// TwinCAT 3 PLC project XPlanarPLC
// ProgramVersion: 3.1.4026.19
// libraries:
//   SPT Base Types, * (Beckhoff Automation LLC)
//   Tc2_Standard, * (Beckhoff Automation GmbH)
//   Tc2_System, * (Beckhoff Automation GmbH)
//   Tc2_Utilities, * (Beckhoff Automation GmbH)
//   Tc3_Mc3PlanarMotion, * (Beckhoff Automation GmbH)
//   Tc3_XPlanarUtility, * (Beckhoff Automation GmbH)
//   XPlanarApplication, * (Beckhoff Automation LLC)
// project tree:
//   DUTs/Estop/ E_EStop.TcDUT, ST_EstopIO.TcDUT, U_Estop.TcDUT
//   DUTs/ E_DemoStep.TcDUT, ST_Point.TcDUT
//   DUTs/Selector switch/ E_SelectorSwitchPos.TcDUT, ST_SelectorSwitchIO.TcDUT, U_SelectorSwitch.TcDUT
//   / PlcTask.TcTTO
//   POUs/ F_SetAllMoversMovement.TcPOU, F_SetAllMoversRotation.TcPOU, MAIN.TcPOU
//   POUs/Pushbuttons/ FB_Pushbutton.TcPOU, LED_Color_Enum.TcDUT, Pushbutton_Enum.TcDUT
// real-time tasks:
//   TASK PlcTask: cycle T#10ms, priority 20, ADS port 350
//   TASK XPlanar Task3: cycle T#250us, priority 1, ADS port 351
//   TASK MC-Task (MET): cycle T#2ms, priority 2, ADS port 352
//   TASK MC-Task (MPT): cycle T#10ms, priority 3, ADS port 353
//   TASK Job Task: cycle default, priority 4
// I/O:
//   DEVICE Device 3 (EtherCAT), AmsNetId 172.18.232.79.4.1
//     Box 6 (PS2001-2420) [PS2001-2420-1001 Power supply (24V, 20A, 1-phase)]
//     Box 5 (EP2339-0003) [EP2339-0003 16 Ch. Dig. Input/Output 24V, 0,5A, 10-Pole Plug Connector]
//   DEVICE Device 1 (EtherCAT), AmsNetId 172.18.232.79.2.1
//     Term 1 (APS4322-7000) [APS4322-7000 Drive]
//       Term 2 (APS4322-5000) [APS4322-5000 Feedback]
//     Term 3 (APS4322-7000) [APS4322-7000 Drive]
//       Term 4 (APS4322-5000) [APS4322-5000 Feedback]
// variable links:
//   Device 1 (EtherCAT) <-> TcCOM Objects/XPlanar/Part1/Tile1
//     Term 3 (APS4322-7000)/APS Comm Inputs/CommStatusWord <-> Data Pointer/MoverCommStatusWord
//     Term 3 (APS4322-7000)/APS Comm Inputs/Data {1..4} <-> Data Pointer/MoverCommDataIn[{0..3}]  (4 links)
//     Term 3 (APS4322-7000)/APS Comm Outputs/CommControlWord <-> Data Pointer/MoverCommControlWord
//     Term 3 (APS4322-7000)/APS Comm Outputs/Data 1 <-> Data Pointer/MoverCommDataOut
//     Term 3 (APS4322-7000)/APS Diagdata/DC Link Voltage <-> Data Pointer/DcLinkVoltage
//     Term 3 (APS4322-7000)/APS Diagdata/Power supply current <-> Data Pointer/PowerSupplyCurrent
//     Term 3 (APS4322-7000)/APS Inputs/StatusWord <-> Data Pointer/PowerUnitStatusWord
//     Term 3 (APS4322-7000)/APS Outputs/ControlWord <-> Data Pointer/PowerUnitControlWord
//     Term 3 (APS4322-7000)/APS Outputs/Current D 0X0 <-> Data Pointer/DCurrentSetPoints[0]
//     Term 3 (APS4322-7000)/APS Outputs/Current D 0X1 <-> Data Pointer/DCurrentSetPoints[1]
//     Term 3 (APS4322-7000)/APS Outputs/Current D 0X2 <-> Data Pointer/DCurrentSetPoints[2]
//     Term 3 (APS4322-7000)/APS Outputs/Current D 1X0 <-> Data Pointer/DCurrentSetPoints[6]
//     Term 3 (APS4322-7000)/APS Outputs/Current D 1X1 <-> Data Pointer/DCurrentSetPoints[7]
//     Term 3 (APS4322-7000)/APS Outputs/Current D 1X2 <-> Data Pointer/DCurrentSetPoints[8]
//     Term 3 (APS4322-7000)/APS Outputs/Current D 2X0 <-> Data Pointer/DCurrentSetPoints[12]
//     Term 3 (APS4322-7000)/APS Outputs/Current D 2X1 <-> Data Pointer/DCurrentSetPoints[13]
//     Term 3 (APS4322-7000)/APS Outputs/Current D 2X2 <-> Data Pointer/DCurrentSetPoints[14]
//     Term 3 (APS4322-7000)/APS Outputs/Current D 3X0 <-> Data Pointer/DCurrentSetPoints[18]
//     Term 3 (APS4322-7000)/APS Outputs/Current D 3X1 <-> Data Pointer/DCurrentSetPoints[19]
//     Term 3 (APS4322-7000)/APS Outputs/Current D 3X2 <-> Data Pointer/DCurrentSetPoints[20]
//     Term 3 (APS4322-7000)/APS Outputs/Current D 0Y0 <-> Data Pointer/DCurrentSetPoints[3]
//     Term 3 (APS4322-7000)/APS Outputs/Current D 0Y1 <-> Data Pointer/DCurrentSetPoints[4]
//     Term 3 (APS4322-7000)/APS Outputs/Current D 0Y2 <-> Data Pointer/DCurrentSetPoints[5]
//     Term 3 (APS4322-7000)/APS Outputs/Current D 1Y0 <-> Data Pointer/DCurrentSetPoints[9]
//     Term 3 (APS4322-7000)/APS Outputs/Current D 1Y1 <-> Data Pointer/DCurrentSetPoints[10]
//     Term 3 (APS4322-7000)/APS Outputs/Current D 1Y2 <-> Data Pointer/DCurrentSetPoints[11]
//     Term 3 (APS4322-7000)/APS Outputs/Current D 2Y0 <-> Data Pointer/DCurrentSetPoints[15]
//     Term 3 (APS4322-7000)/APS Outputs/Current D 2Y1 <-> Data Pointer/DCurrentSetPoints[16]
//     Term 3 (APS4322-7000)/APS Outputs/Current D 2Y2 <-> Data Pointer/DCurrentSetPoints[17]
//     Term 3 (APS4322-7000)/APS Outputs/Current D 3Y0 <-> Data Pointer/DCurrentSetPoints[21]
//     Term 3 (APS4322-7000)/APS Outputs/Current D 3Y1 <-> Data Pointer/DCurrentSetPoints[22]
//     Term 3 (APS4322-7000)/APS Outputs/Current D 3Y2 <-> Data Pointer/DCurrentSetPoints[23]
//     Term 3 (APS4322-7000)/APS Outputs/Current Q 0X0 <-> Data Pointer/QCurrentSetPoints[0]
//     Term 3 (APS4322-7000)/APS Outputs/Current Q 0X1 <-> Data Pointer/QCurrentSetPoints[1]
//     Term 3 (APS4322-7000)/APS Outputs/Current Q 0X2 <-> Data Pointer/QCurrentSetPoints[2]
//     Term 3 (APS4322-7000)/APS Outputs/Current Q 1X0 <-> Data Pointer/QCurrentSetPoints[6]
//     Term 3 (APS4322-7000)/APS Outputs/Current Q 1X1 <-> Data Pointer/QCurrentSetPoints[7]
//     Term 3 (APS4322-7000)/APS Outputs/Current Q 1X2 <-> Data Pointer/QCurrentSetPoints[8]
//     Term 3 (APS4322-7000)/APS Outputs/Current Q 2X0 <-> Data Pointer/QCurrentSetPoints[12]
//     Term 3 (APS4322-7000)/APS Outputs/Current Q 2X1 <-> Data Pointer/QCurrentSetPoints[13]
//     Term 3 (APS4322-7000)/APS Outputs/Current Q 2X2 <-> Data Pointer/QCurrentSetPoints[14]
//     Term 3 (APS4322-7000)/APS Outputs/Current Q 3X0 <-> Data Pointer/QCurrentSetPoints[18]
//     Term 3 (APS4322-7000)/APS Outputs/Current Q 3X1 <-> Data Pointer/QCurrentSetPoints[19]
//     Term 3 (APS4322-7000)/APS Outputs/Current Q 3X2 <-> Data Pointer/QCurrentSetPoints[20]
//     Term 3 (APS4322-7000)/APS Outputs/Current Q 0Y0 <-> Data Pointer/QCurrentSetPoints[3]
//     Term 3 (APS4322-7000)/APS Outputs/Current Q 0Y1 <-> Data Pointer/QCurrentSetPoints[4]
//     Term 3 (APS4322-7000)/APS Outputs/Current Q 0Y2 <-> Data Pointer/QCurrentSetPoints[5]
//     Term 3 (APS4322-7000)/APS Outputs/Current Q 1Y0 <-> Data Pointer/QCurrentSetPoints[9]
//     Term 3 (APS4322-7000)/APS Outputs/Current Q 1Y1 <-> Data Pointer/QCurrentSetPoints[10]
//     Term 3 (APS4322-7000)/APS Outputs/Current Q 1Y2 <-> Data Pointer/QCurrentSetPoints[11]
//     Term 3 (APS4322-7000)/APS Outputs/Current Q 2Y0 <-> Data Pointer/QCurrentSetPoints[15]
//     Term 3 (APS4322-7000)/APS Outputs/Current Q 2Y1 <-> Data Pointer/QCurrentSetPoints[16]
//     Term 3 (APS4322-7000)/APS Outputs/Current Q 2Y2 <-> Data Pointer/QCurrentSetPoints[17]
//     Term 3 (APS4322-7000)/APS Outputs/Current Q 3Y0 <-> Data Pointer/QCurrentSetPoints[21]
//     Term 3 (APS4322-7000)/APS Outputs/Current Q 3Y1 <-> Data Pointer/QCurrentSetPoints[22]
//     Term 3 (APS4322-7000)/APS Outputs/Current Q 3Y2 <-> Data Pointer/QCurrentSetPoints[23]
//     Term 3 (APS4322-7000)/APS Outputs/PhiE 0X0 <-> Data Pointer/PhiSetPoints[0]
//     Term 3 (APS4322-7000)/APS Outputs/PhiE 0X1 <-> Data Pointer/PhiSetPoints[1]
//     Term 3 (APS4322-7000)/APS Outputs/PhiE 0X2 <-> Data Pointer/PhiSetPoints[2]
//     Term 3 (APS4322-7000)/APS Outputs/PhiE 1X0 <-> Data Pointer/PhiSetPoints[6]
//     Term 3 (APS4322-7000)/APS Outputs/PhiE 1X1 <-> Data Pointer/PhiSetPoints[7]
//     Term 3 (APS4322-7000)/APS Outputs/PhiE 1X2 <-> Data Pointer/PhiSetPoints[8]
//     Term 3 (APS4322-7000)/APS Outputs/PhiE 2X0 <-> Data Pointer/PhiSetPoints[12]
//     Term 3 (APS4322-7000)/APS Outputs/PhiE 2X1 <-> Data Pointer/PhiSetPoints[13]
//     Term 3 (APS4322-7000)/APS Outputs/PhiE 2X2 <-> Data Pointer/PhiSetPoints[14]
//     Term 3 (APS4322-7000)/APS Outputs/PhiE 3X0 <-> Data Pointer/PhiSetPoints[18]
//     Term 3 (APS4322-7000)/APS Outputs/PhiE 3X1 <-> Data Pointer/PhiSetPoints[19]
//     Term 3 (APS4322-7000)/APS Outputs/PhiE 3X2 <-> Data Pointer/PhiSetPoints[20]
//     Term 3 (APS4322-7000)/APS Outputs/PhiE 0Y0 <-> Data Pointer/PhiSetPoints[3]
//     Term 3 (APS4322-7000)/APS Outputs/PhiE 0Y1 <-> Data Pointer/PhiSetPoints[4]
//     Term 3 (APS4322-7000)/APS Outputs/PhiE 0Y2 <-> Data Pointer/PhiSetPoints[5]
//     Term 3 (APS4322-7000)/APS Outputs/PhiE 1Y0 <-> Data Pointer/PhiSetPoints[9]
//     Term 3 (APS4322-7000)/APS Outputs/PhiE 1Y1 <-> Data Pointer/PhiSetPoints[10]
//     Term 3 (APS4322-7000)/APS Outputs/PhiE 1Y2 <-> Data Pointer/PhiSetPoints[11]
//     Term 3 (APS4322-7000)/APS Outputs/PhiE 2Y0 <-> Data Pointer/PhiSetPoints[15]
//     Term 3 (APS4322-7000)/APS Outputs/PhiE 2Y1 <-> Data Pointer/PhiSetPoints[16]
//     Term 3 (APS4322-7000)/APS Outputs/PhiE 2Y2 <-> Data Pointer/PhiSetPoints[17]
//     Term 3 (APS4322-7000)/APS Outputs/PhiE 3Y0 <-> Data Pointer/PhiSetPoints[21]
//     Term 3 (APS4322-7000)/APS Outputs/PhiE 3Y1 <-> Data Pointer/PhiSetPoints[22]
//     Term 3 (APS4322-7000)/APS Outputs/PhiE 3Y2 <-> Data Pointer/PhiSetPoints[23]
//     Term 3 (APS4322-7000)/Term 4 (APS4322-5000)/FB Inputs/A{0..8 step 2} X-Field <-> Data Pointer/HallSensorFieldsXYZ[{0..12 step 3}]  (5 links)
//     Term 3 (APS4322-7000)/Term 4 (APS4322-5000)/FB Inputs/A{0..8 step 2} Y-Field <-> Data Pointer/HallSensorFieldsXYZ[{1..13 step 3}]  (5 links)
//     Term 3 (APS4322-7000)/Term 4 (APS4322-5000)/FB Inputs/A{0..8 step 2} Z-Field <-> Data Pointer/HallSensorFieldsXYZ[{2..14 step 3}]  (5 links)
//     Term 3 (APS4322-7000)/Term 4 (APS4322-5000)/FB Inputs/B{1..9 step 2} X-Field <-> Data Pointer/HallSensorFieldsXYZ[{15..27 step 3}]  (5 links)
//     Term 3 (APS4322-7000)/Term 4 (APS4322-5000)/FB Inputs/B{1..9 step 2} Y-Field <-> Data Pointer/HallSensorFieldsXYZ[{16..28 step 3}]  (5 links)
//     Term 3 (APS4322-7000)/Term 4 (APS4322-5000)/FB Inputs/B{1..9 step 2} Z-Field <-> Data Pointer/HallSensorFieldsXYZ[{17..29 step 3}]  (5 links)
//     Term 3 (APS4322-7000)/Term 4 (APS4322-5000)/FB Inputs/C{0..8 step 2} X-Field <-> Data Pointer/HallSensorFieldsXYZ[{30..42 step 3}]  (5 links)
//     Term 3 (APS4322-7000)/Term 4 (APS4322-5000)/FB Inputs/C{0..8 step 2} Y-Field <-> Data Pointer/HallSensorFieldsXYZ[{31..43 step 3}]  (5 links)
//     Term 3 (APS4322-7000)/Term 4 (APS4322-5000)/FB Inputs/C{0..8 step 2} Z-Field <-> Data Pointer/HallSensorFieldsXYZ[{32..44 step 3}]  (5 links)
//     Term 3 (APS4322-7000)/Term 4 (APS4322-5000)/FB Inputs/D{1..9 step 2} X-Field <-> Data Pointer/HallSensorFieldsXYZ[{45..57 step 3}]  (5 links)
//     Term 3 (APS4322-7000)/Term 4 (APS4322-5000)/FB Inputs/D{1..9 step 2} Y-Field <-> Data Pointer/HallSensorFieldsXYZ[{46..58 step 3}]  (5 links)
//     Term 3 (APS4322-7000)/Term 4 (APS4322-5000)/FB Inputs/D{1..9 step 2} Z-Field <-> Data Pointer/HallSensorFieldsXYZ[{47..59 step 3}]  (5 links)
//     Term 3 (APS4322-7000)/Term 4 (APS4322-5000)/FB Inputs/E{0..8 step 2} X-Field <-> Data Pointer/HallSensorFieldsXYZ[{60..72 step 3}]  (5 links)
//     Term 3 (APS4322-7000)/Term 4 (APS4322-5000)/FB Inputs/E{0..8 step 2} Y-Field <-> Data Pointer/HallSensorFieldsXYZ[{61..73 step 3}]  (5 links)
//     Term 3 (APS4322-7000)/Term 4 (APS4322-5000)/FB Inputs/E{0..8 step 2} Z-Field <-> Data Pointer/HallSensorFieldsXYZ[{62..74 step 3}]  (5 links)
//     Term 3 (APS4322-7000)/Term 4 (APS4322-5000)/FB Inputs/F{1..9 step 2} X-Field <-> Data Pointer/HallSensorFieldsXYZ[{75..87 step 3}]  (5 links)
//     Term 3 (APS4322-7000)/Term 4 (APS4322-5000)/FB Inputs/F{1..9 step 2} Y-Field <-> Data Pointer/HallSensorFieldsXYZ[{76..88 step 3}]  (5 links)
//     Term 3 (APS4322-7000)/Term 4 (APS4322-5000)/FB Inputs/F{1..9 step 2} Z-Field <-> Data Pointer/HallSensorFieldsXYZ[{77..89 step 3}]  (5 links)
//     Term 3 (APS4322-7000)/Term 4 (APS4322-5000)/FB Inputs/G{0..8 step 2} X-Field <-> Data Pointer/HallSensorFieldsXYZ[{90..102 step 3}]  (5 links)
//     Term 3 (APS4322-7000)/Term 4 (APS4322-5000)/FB Inputs/G{0..8 step 2} Y-Field <-> Data Pointer/HallSensorFieldsXYZ[{91..103 step 3}]  (5 links)
//     Term 3 (APS4322-7000)/Term 4 (APS4322-5000)/FB Inputs/G{0..8 step 2} Z-Field <-> Data Pointer/HallSensorFieldsXYZ[{92..104 step 3}]  (5 links)
//     Term 3 (APS4322-7000)/Term 4 (APS4322-5000)/FB Inputs/H{1..9 step 2} X-Field <-> Data Pointer/HallSensorFieldsXYZ[{105..117 step 3}]  (5 links)
//     Term 3 (APS4322-7000)/Term 4 (APS4322-5000)/FB Inputs/H{1..9 step 2} Y-Field <-> Data Pointer/HallSensorFieldsXYZ[{106..118 step 3}]  (5 links)
//     Term 3 (APS4322-7000)/Term 4 (APS4322-5000)/FB Inputs/H{1..9 step 2} Z-Field <-> Data Pointer/HallSensorFieldsXYZ[{107..119 step 3}]  (5 links)
//     Term 3 (APS4322-7000)/Term 4 (APS4322-5000)/FB Inputs/I{0..8 step 2} X-Field <-> Data Pointer/HallSensorFieldsXYZ[{120..132 step 3}]  (5 links)
//     Term 3 (APS4322-7000)/Term 4 (APS4322-5000)/FB Inputs/I{0..8 step 2} Y-Field <-> Data Pointer/HallSensorFieldsXYZ[{121..133 step 3}]  (5 links)
//     Term 3 (APS4322-7000)/Term 4 (APS4322-5000)/FB Inputs/I{0..8 step 2} Z-Field <-> Data Pointer/HallSensorFieldsXYZ[{122..134 step 3}]  (5 links)
//     Term 3 (APS4322-7000)/Term 4 (APS4322-5000)/FB Inputs/J{1..9 step 2} X-Field <-> Data Pointer/HallSensorFieldsXYZ[{135..147 step 3}]  (5 links)
//     Term 3 (APS4322-7000)/Term 4 (APS4322-5000)/FB Inputs/J{1..9 step 2} Y-Field <-> Data Pointer/HallSensorFieldsXYZ[{136..148 step 3}]  (5 links)
//     Term 3 (APS4322-7000)/Term 4 (APS4322-5000)/FB Inputs/J{1..9 step 2} Z-Field <-> Data Pointer/HallSensorFieldsXYZ[{137..149 step 3}]  (5 links)
//     Term 3 (APS4322-7000)/Term 4 (APS4322-5000)/FB Inputs/Status <-> Data Pointer/FeedbackStatus
//   Device 1 (EtherCAT) <-> TcCOM Objects/XPlanar/Part1/Tile2
//     Term 1 (APS4322-7000)/APS Comm Inputs/CommStatusWord <-> Data Pointer/MoverCommStatusWord
//     Term 1 (APS4322-7000)/APS Comm Inputs/Data {1..4} <-> Data Pointer/MoverCommDataIn[{0..3}]  (4 links)
//     Term 1 (APS4322-7000)/APS Comm Outputs/CommControlWord <-> Data Pointer/MoverCommControlWord
//     Term 1 (APS4322-7000)/APS Comm Outputs/Data 1 <-> Data Pointer/MoverCommDataOut
//     Term 1 (APS4322-7000)/APS Diagdata/DC Link Voltage <-> Data Pointer/DcLinkVoltage
//     Term 1 (APS4322-7000)/APS Diagdata/Power supply current <-> Data Pointer/PowerSupplyCurrent
//     Term 1 (APS4322-7000)/APS Inputs/StatusWord <-> Data Pointer/PowerUnitStatusWord
//     Term 1 (APS4322-7000)/APS Outputs/ControlWord <-> Data Pointer/PowerUnitControlWord
//     Term 1 (APS4322-7000)/APS Outputs/Current D 0X0 <-> Data Pointer/DCurrentSetPoints[0]
//     Term 1 (APS4322-7000)/APS Outputs/Current D 0X1 <-> Data Pointer/DCurrentSetPoints[1]
//     Term 1 (APS4322-7000)/APS Outputs/Current D 0X2 <-> Data Pointer/DCurrentSetPoints[2]
//     Term 1 (APS4322-7000)/APS Outputs/Current D 1X0 <-> Data Pointer/DCurrentSetPoints[6]
//     Term 1 (APS4322-7000)/APS Outputs/Current D 1X1 <-> Data Pointer/DCurrentSetPoints[7]
//     Term 1 (APS4322-7000)/APS Outputs/Current D 1X2 <-> Data Pointer/DCurrentSetPoints[8]
//     Term 1 (APS4322-7000)/APS Outputs/Current D 2X0 <-> Data Pointer/DCurrentSetPoints[12]
//     Term 1 (APS4322-7000)/APS Outputs/Current D 2X1 <-> Data Pointer/DCurrentSetPoints[13]
//     Term 1 (APS4322-7000)/APS Outputs/Current D 2X2 <-> Data Pointer/DCurrentSetPoints[14]
//     Term 1 (APS4322-7000)/APS Outputs/Current D 3X0 <-> Data Pointer/DCurrentSetPoints[18]
//     Term 1 (APS4322-7000)/APS Outputs/Current D 3X1 <-> Data Pointer/DCurrentSetPoints[19]
//     Term 1 (APS4322-7000)/APS Outputs/Current D 3X2 <-> Data Pointer/DCurrentSetPoints[20]
//     Term 1 (APS4322-7000)/APS Outputs/Current D 0Y0 <-> Data Pointer/DCurrentSetPoints[3]
//     Term 1 (APS4322-7000)/APS Outputs/Current D 0Y1 <-> Data Pointer/DCurrentSetPoints[4]
//     Term 1 (APS4322-7000)/APS Outputs/Current D 0Y2 <-> Data Pointer/DCurrentSetPoints[5]
//     Term 1 (APS4322-7000)/APS Outputs/Current D 1Y0 <-> Data Pointer/DCurrentSetPoints[9]
//     Term 1 (APS4322-7000)/APS Outputs/Current D 1Y1 <-> Data Pointer/DCurrentSetPoints[10]
//     Term 1 (APS4322-7000)/APS Outputs/Current D 1Y2 <-> Data Pointer/DCurrentSetPoints[11]
//     Term 1 (APS4322-7000)/APS Outputs/Current D 2Y0 <-> Data Pointer/DCurrentSetPoints[15]
//     Term 1 (APS4322-7000)/APS Outputs/Current D 2Y1 <-> Data Pointer/DCurrentSetPoints[16]
//     Term 1 (APS4322-7000)/APS Outputs/Current D 2Y2 <-> Data Pointer/DCurrentSetPoints[17]
//     Term 1 (APS4322-7000)/APS Outputs/Current D 3Y0 <-> Data Pointer/DCurrentSetPoints[21]
//     Term 1 (APS4322-7000)/APS Outputs/Current D 3Y1 <-> Data Pointer/DCurrentSetPoints[22]
//     Term 1 (APS4322-7000)/APS Outputs/Current D 3Y2 <-> Data Pointer/DCurrentSetPoints[23]
//     Term 1 (APS4322-7000)/APS Outputs/Current Q 0X0 <-> Data Pointer/QCurrentSetPoints[0]
//     Term 1 (APS4322-7000)/APS Outputs/Current Q 0X1 <-> Data Pointer/QCurrentSetPoints[1]
//     Term 1 (APS4322-7000)/APS Outputs/Current Q 0X2 <-> Data Pointer/QCurrentSetPoints[2]
//     Term 1 (APS4322-7000)/APS Outputs/Current Q 1X0 <-> Data Pointer/QCurrentSetPoints[6]
//     Term 1 (APS4322-7000)/APS Outputs/Current Q 1X1 <-> Data Pointer/QCurrentSetPoints[7]
//     Term 1 (APS4322-7000)/APS Outputs/Current Q 1X2 <-> Data Pointer/QCurrentSetPoints[8]
//     Term 1 (APS4322-7000)/APS Outputs/Current Q 2X0 <-> Data Pointer/QCurrentSetPoints[12]
//     Term 1 (APS4322-7000)/APS Outputs/Current Q 2X1 <-> Data Pointer/QCurrentSetPoints[13]
//     Term 1 (APS4322-7000)/APS Outputs/Current Q 2X2 <-> Data Pointer/QCurrentSetPoints[14]
//     Term 1 (APS4322-7000)/APS Outputs/Current Q 3X0 <-> Data Pointer/QCurrentSetPoints[18]
//     Term 1 (APS4322-7000)/APS Outputs/Current Q 3X1 <-> Data Pointer/QCurrentSetPoints[19]
//     Term 1 (APS4322-7000)/APS Outputs/Current Q 3X2 <-> Data Pointer/QCurrentSetPoints[20]
//     Term 1 (APS4322-7000)/APS Outputs/Current Q 0Y0 <-> Data Pointer/QCurrentSetPoints[3]
//     Term 1 (APS4322-7000)/APS Outputs/Current Q 0Y1 <-> Data Pointer/QCurrentSetPoints[4]
//     Term 1 (APS4322-7000)/APS Outputs/Current Q 0Y2 <-> Data Pointer/QCurrentSetPoints[5]
//     Term 1 (APS4322-7000)/APS Outputs/Current Q 1Y0 <-> Data Pointer/QCurrentSetPoints[9]
//     Term 1 (APS4322-7000)/APS Outputs/Current Q 1Y1 <-> Data Pointer/QCurrentSetPoints[10]
//     Term 1 (APS4322-7000)/APS Outputs/Current Q 1Y2 <-> Data Pointer/QCurrentSetPoints[11]
//     Term 1 (APS4322-7000)/APS Outputs/Current Q 2Y0 <-> Data Pointer/QCurrentSetPoints[15]
//     Term 1 (APS4322-7000)/APS Outputs/Current Q 2Y1 <-> Data Pointer/QCurrentSetPoints[16]
//     Term 1 (APS4322-7000)/APS Outputs/Current Q 2Y2 <-> Data Pointer/QCurrentSetPoints[17]
//     Term 1 (APS4322-7000)/APS Outputs/Current Q 3Y0 <-> Data Pointer/QCurrentSetPoints[21]
//     Term 1 (APS4322-7000)/APS Outputs/Current Q 3Y1 <-> Data Pointer/QCurrentSetPoints[22]
//     Term 1 (APS4322-7000)/APS Outputs/Current Q 3Y2 <-> Data Pointer/QCurrentSetPoints[23]
//     Term 1 (APS4322-7000)/APS Outputs/PhiE 0X0 <-> Data Pointer/PhiSetPoints[0]
//     Term 1 (APS4322-7000)/APS Outputs/PhiE 0X1 <-> Data Pointer/PhiSetPoints[1]
//     Term 1 (APS4322-7000)/APS Outputs/PhiE 0X2 <-> Data Pointer/PhiSetPoints[2]
//     Term 1 (APS4322-7000)/APS Outputs/PhiE 1X0 <-> Data Pointer/PhiSetPoints[6]
//     Term 1 (APS4322-7000)/APS Outputs/PhiE 1X1 <-> Data Pointer/PhiSetPoints[7]
//     Term 1 (APS4322-7000)/APS Outputs/PhiE 1X2 <-> Data Pointer/PhiSetPoints[8]
//     Term 1 (APS4322-7000)/APS Outputs/PhiE 2X0 <-> Data Pointer/PhiSetPoints[12]
//     Term 1 (APS4322-7000)/APS Outputs/PhiE 2X1 <-> Data Pointer/PhiSetPoints[13]
//     Term 1 (APS4322-7000)/APS Outputs/PhiE 2X2 <-> Data Pointer/PhiSetPoints[14]
//     Term 1 (APS4322-7000)/APS Outputs/PhiE 3X0 <-> Data Pointer/PhiSetPoints[18]
//     Term 1 (APS4322-7000)/APS Outputs/PhiE 3X1 <-> Data Pointer/PhiSetPoints[19]
//     Term 1 (APS4322-7000)/APS Outputs/PhiE 3X2 <-> Data Pointer/PhiSetPoints[20]
//     Term 1 (APS4322-7000)/APS Outputs/PhiE 0Y0 <-> Data Pointer/PhiSetPoints[3]
//     Term 1 (APS4322-7000)/APS Outputs/PhiE 0Y1 <-> Data Pointer/PhiSetPoints[4]
//     Term 1 (APS4322-7000)/APS Outputs/PhiE 0Y2 <-> Data Pointer/PhiSetPoints[5]
//     Term 1 (APS4322-7000)/APS Outputs/PhiE 1Y0 <-> Data Pointer/PhiSetPoints[9]
//     Term 1 (APS4322-7000)/APS Outputs/PhiE 1Y1 <-> Data Pointer/PhiSetPoints[10]
//     Term 1 (APS4322-7000)/APS Outputs/PhiE 1Y2 <-> Data Pointer/PhiSetPoints[11]
//     Term 1 (APS4322-7000)/APS Outputs/PhiE 2Y0 <-> Data Pointer/PhiSetPoints[15]
//     Term 1 (APS4322-7000)/APS Outputs/PhiE 2Y1 <-> Data Pointer/PhiSetPoints[16]
//     Term 1 (APS4322-7000)/APS Outputs/PhiE 2Y2 <-> Data Pointer/PhiSetPoints[17]
//     Term 1 (APS4322-7000)/APS Outputs/PhiE 3Y0 <-> Data Pointer/PhiSetPoints[21]
//     Term 1 (APS4322-7000)/APS Outputs/PhiE 3Y1 <-> Data Pointer/PhiSetPoints[22]
//     Term 1 (APS4322-7000)/APS Outputs/PhiE 3Y2 <-> Data Pointer/PhiSetPoints[23]
//     Term 1 (APS4322-7000)/Term 2 (APS4322-5000)/FB Inputs/A{0..8 step 2} X-Field <-> Data Pointer/HallSensorFieldsXYZ[{0..12 step 3}]  (5 links)
//     Term 1 (APS4322-7000)/Term 2 (APS4322-5000)/FB Inputs/A{0..8 step 2} Y-Field <-> Data Pointer/HallSensorFieldsXYZ[{1..13 step 3}]  (5 links)
//     Term 1 (APS4322-7000)/Term 2 (APS4322-5000)/FB Inputs/A{0..8 step 2} Z-Field <-> Data Pointer/HallSensorFieldsXYZ[{2..14 step 3}]  (5 links)
//     Term 1 (APS4322-7000)/Term 2 (APS4322-5000)/FB Inputs/B{1..9 step 2} X-Field <-> Data Pointer/HallSensorFieldsXYZ[{15..27 step 3}]  (5 links)
//     Term 1 (APS4322-7000)/Term 2 (APS4322-5000)/FB Inputs/B{1..9 step 2} Y-Field <-> Data Pointer/HallSensorFieldsXYZ[{16..28 step 3}]  (5 links)
//     Term 1 (APS4322-7000)/Term 2 (APS4322-5000)/FB Inputs/B{1..9 step 2} Z-Field <-> Data Pointer/HallSensorFieldsXYZ[{17..29 step 3}]  (5 links)
//     Term 1 (APS4322-7000)/Term 2 (APS4322-5000)/FB Inputs/C{0..8 step 2} X-Field <-> Data Pointer/HallSensorFieldsXYZ[{30..42 step 3}]  (5 links)
//     Term 1 (APS4322-7000)/Term 2 (APS4322-5000)/FB Inputs/C{0..8 step 2} Y-Field <-> Data Pointer/HallSensorFieldsXYZ[{31..43 step 3}]  (5 links)
//     Term 1 (APS4322-7000)/Term 2 (APS4322-5000)/FB Inputs/C{0..8 step 2} Z-Field <-> Data Pointer/HallSensorFieldsXYZ[{32..44 step 3}]  (5 links)
//     Term 1 (APS4322-7000)/Term 2 (APS4322-5000)/FB Inputs/D{1..9 step 2} X-Field <-> Data Pointer/HallSensorFieldsXYZ[{45..57 step 3}]  (5 links)
//     Term 1 (APS4322-7000)/Term 2 (APS4322-5000)/FB Inputs/D{1..9 step 2} Y-Field <-> Data Pointer/HallSensorFieldsXYZ[{46..58 step 3}]  (5 links)
//     Term 1 (APS4322-7000)/Term 2 (APS4322-5000)/FB Inputs/D{1..9 step 2} Z-Field <-> Data Pointer/HallSensorFieldsXYZ[{47..59 step 3}]  (5 links)
//     Term 1 (APS4322-7000)/Term 2 (APS4322-5000)/FB Inputs/E{0..8 step 2} X-Field <-> Data Pointer/HallSensorFieldsXYZ[{60..72 step 3}]  (5 links)
//     Term 1 (APS4322-7000)/Term 2 (APS4322-5000)/FB Inputs/E{0..8 step 2} Y-Field <-> Data Pointer/HallSensorFieldsXYZ[{61..73 step 3}]  (5 links)
//     Term 1 (APS4322-7000)/Term 2 (APS4322-5000)/FB Inputs/E{0..8 step 2} Z-Field <-> Data Pointer/HallSensorFieldsXYZ[{62..74 step 3}]  (5 links)
//     Term 1 (APS4322-7000)/Term 2 (APS4322-5000)/FB Inputs/F{1..9 step 2} X-Field <-> Data Pointer/HallSensorFieldsXYZ[{75..87 step 3}]  (5 links)
//     Term 1 (APS4322-7000)/Term 2 (APS4322-5000)/FB Inputs/F{1..9 step 2} Y-Field <-> Data Pointer/HallSensorFieldsXYZ[{76..88 step 3}]  (5 links)
//     Term 1 (APS4322-7000)/Term 2 (APS4322-5000)/FB Inputs/F{1..9 step 2} Z-Field <-> Data Pointer/HallSensorFieldsXYZ[{77..89 step 3}]  (5 links)
//     Term 1 (APS4322-7000)/Term 2 (APS4322-5000)/FB Inputs/G{0..8 step 2} X-Field <-> Data Pointer/HallSensorFieldsXYZ[{90..102 step 3}]  (5 links)
//     Term 1 (APS4322-7000)/Term 2 (APS4322-5000)/FB Inputs/G{0..8 step 2} Y-Field <-> Data Pointer/HallSensorFieldsXYZ[{91..103 step 3}]  (5 links)
//     Term 1 (APS4322-7000)/Term 2 (APS4322-5000)/FB Inputs/G{0..8 step 2} Z-Field <-> Data Pointer/HallSensorFieldsXYZ[{92..104 step 3}]  (5 links)
//     Term 1 (APS4322-7000)/Term 2 (APS4322-5000)/FB Inputs/H{1..9 step 2} X-Field <-> Data Pointer/HallSensorFieldsXYZ[{105..117 step 3}]  (5 links)
//     Term 1 (APS4322-7000)/Term 2 (APS4322-5000)/FB Inputs/H{1..9 step 2} Y-Field <-> Data Pointer/HallSensorFieldsXYZ[{106..118 step 3}]  (5 links)
//     Term 1 (APS4322-7000)/Term 2 (APS4322-5000)/FB Inputs/H{1..9 step 2} Z-Field <-> Data Pointer/HallSensorFieldsXYZ[{107..119 step 3}]  (5 links)
//     Term 1 (APS4322-7000)/Term 2 (APS4322-5000)/FB Inputs/I{0..8 step 2} X-Field <-> Data Pointer/HallSensorFieldsXYZ[{120..132 step 3}]  (5 links)
//     Term 1 (APS4322-7000)/Term 2 (APS4322-5000)/FB Inputs/I{0..8 step 2} Y-Field <-> Data Pointer/HallSensorFieldsXYZ[{121..133 step 3}]  (5 links)
//     Term 1 (APS4322-7000)/Term 2 (APS4322-5000)/FB Inputs/I{0..8 step 2} Z-Field <-> Data Pointer/HallSensorFieldsXYZ[{122..134 step 3}]  (5 links)
//     Term 1 (APS4322-7000)/Term 2 (APS4322-5000)/FB Inputs/J{1..9 step 2} X-Field <-> Data Pointer/HallSensorFieldsXYZ[{135..147 step 3}]  (5 links)
//     Term 1 (APS4322-7000)/Term 2 (APS4322-5000)/FB Inputs/J{1..9 step 2} Y-Field <-> Data Pointer/HallSensorFieldsXYZ[{136..148 step 3}]  (5 links)
//     Term 1 (APS4322-7000)/Term 2 (APS4322-5000)/FB Inputs/J{1..9 step 2} Z-Field <-> Data Pointer/HallSensorFieldsXYZ[{137..149 step 3}]  (5 links)
//     Term 1 (APS4322-7000)/Term 2 (APS4322-5000)/FB Inputs/Status <-> Data Pointer/FeedbackStatus
//   TcCOM Objects/XPlanar/Mover4220_1 <-> XPlanar MC Project/Axes/Mover4220_1
//     InputsFromNC3/NC3ToHW <-> McToIo/STD
//     OutputsToNC3/HWToNC3 <-> IoToMc/STD
//   TcCOM Objects/XPlanar/Mover4220_2 <-> XPlanar MC Project/Axes/Mover4220_2
//     InputsFromNC3/NC3ToHW <-> McToIo/STD
//     OutputsToNC3/HWToNC3 <-> IoToMc/STD
//   (this object) <-> Device 3 (EtherCAT)/Box 5 (EP2339-0003)
//     PlcTask Inputs/MAIN.PushButton[0].Pressed <-> DI Inputs Channel 1/Input 4
//     PlcTask Inputs/MAIN.PushButton[1].Pressed <-> DI Inputs Channel 1/Input 8
//     PlcTask Inputs/MAIN.PushButton[2].Pressed <-> DI Inputs Channel 2/Input 4
//     PlcTask Inputs/MAIN.PushButton[3].Pressed <-> DI Inputs Channel 2/Input 8
//     PlcTask Outputs/MAIN.PushButton[0].LED_Blue <-> DO Outputs Channel 1/Output 3
//     PlcTask Outputs/MAIN.PushButton[1].LED_Blue <-> DO Outputs Channel 1/Output 7
//     PlcTask Outputs/MAIN.PushButton[2].LED_Blue <-> DO Outputs Channel 2/Output 3
//     PlcTask Outputs/MAIN.PushButton[3].LED_Blue <-> DO Outputs Channel 2/Output 7
//     PlcTask Outputs/MAIN.PushButton[0].LED_Green <-> DO Outputs Channel 1/Output 2
//     PlcTask Outputs/MAIN.PushButton[1].LED_Green <-> DO Outputs Channel 1/Output 6
//     PlcTask Outputs/MAIN.PushButton[2].LED_Green <-> DO Outputs Channel 2/Output 2
//     PlcTask Outputs/MAIN.PushButton[3].LED_Green <-> DO Outputs Channel 2/Output 6
//     PlcTask Outputs/MAIN.PushButton[0].LED_Red <-> DO Outputs Channel 1/Output 1
//     PlcTask Outputs/MAIN.PushButton[1].LED_Red <-> DO Outputs Channel 1/Output 5
//     PlcTask Outputs/MAIN.PushButton[2].LED_Red <-> DO Outputs Channel 2/Output 1
//     PlcTask Outputs/MAIN.PushButton[3].LED_Red <-> DO Outputs Channel 2/Output 5
//   (this object) <-> XPlanar MC Project/Axes/Mover4220_1
//     PlcTask Inputs/MAIN.Mover1._Mover.MCTOPLC/ACT <-> McToPlc/ACT
//     PlcTask Inputs/MAIN.Mover1._Mover.MCTOPLC/COORDMODE <-> McToPlc/COORDMODE
//     PlcTask Inputs/MAIN.Mover1._Mover.MCTOPLC/SET <-> McToPlc/SET
//     PlcTask Inputs/MAIN.Mover1._Mover.MCTOPLC/SETONTRACK <-> McToPlc/SETONTRACK
//     PlcTask Inputs/MAIN.Mover1._Mover.MCTOPLC/STD <-> McToPlc/STD
//     PlcTask Outputs/MAIN.Mover1._Mover.PLCTOMC/STD <-> PlcToMc/STD
//   (this object) <-> XPlanar MC Project/Axes/Mover4220_2
//     PlcTask Inputs/MAIN.Mover2._Mover.MCTOPLC/ACT <-> McToPlc/ACT
//     PlcTask Inputs/MAIN.Mover2._Mover.MCTOPLC/COORDMODE <-> McToPlc/COORDMODE
//     PlcTask Inputs/MAIN.Mover2._Mover.MCTOPLC/SET <-> McToPlc/SET
//     PlcTask Inputs/MAIN.Mover2._Mover.MCTOPLC/SETONTRACK <-> McToPlc/SETONTRACK
//     PlcTask Inputs/MAIN.Mover2._Mover.MCTOPLC/STD <-> McToPlc/STD
//     PlcTask Outputs/MAIN.Mover2._Mover.PLCTOMC/STD <-> PlcToMc/STD
//   (this object) <-> XPlanar MC Project/Groups/Environment
//     PlcTask Inputs/XPlanar.Environment.MCTOPLC_STD <-> McToPlc/STD
//   (this object) <-> XPlanar MC Project/Groups/Track1
//     PlcTask Inputs/MAIN.Track1._Track.MCTOPLC_STD <-> McToPlc/STD
//   (this object) <-> XPlanar MC Project/Groups/XPlanar
//     PlcTask Inputs/XPlanar.Group.MCTOPLC_STD <-> McToPlc/STD

CONFIGURATION XPlanarPLC
    RESOURCE PLC ON TwinCAT3
        TASK PlcTask(INTERVAL := T#10ms, PRIORITY := 20);
        PROGRAM MAIN WITH PlcTask : MAIN;
    END_RESOURCE
END_CONFIGURATION

// ---- DUTs/Estop/E_EStop.TcDUT
{attribute 'qualified_only'}
{attribute 'strict'}
{attribute 'to_string'}
TYPE E_EStop :
(
	Activated		:=0,
	Normallyclosed 	:=3

)BYTE;
END_TYPE

// ---- DUTs/Estop/ST_EstopIO.TcDUT
TYPE ST_EstopIO :
STRUCT
	ch1	AT%I* 	:BIT;
	Ch2	AT%I*	:BIT;	
END_STRUCT
END_TYPE

// ---- DUTs/Estop/U_Estop.TcDUT
TYPE U_Estop :
UNION
	Pos	:E_EStop;	
	IO 	:ST_EstopIO;
END_UNION
END_TYPE

// ---- DUTs/E_DemoStep.TcDUT
{attribute 'qualified_only'}
{attribute 'strict'}
{attribute 'to_string'}
TYPE E_DemoStep :
(
	Init := 0,
	WaitForSwitch,
	DetectMovers,
	SortMovers,	
	Enabling,
	SquareUpMovers,
	MoveToSeqenceStartPos,
	JoinTrack,
	FigureEight,
	LeaveTrack,
	GoToOpositeCorner,
	FlyBy,
	MoveAroundPerimeter,
	MoveToCenterOfTiles,
	RotateInverse,
	Spin,
	Lift,
	Tilt,
	Disable
);
END_TYPE

// ---- DUTs/Selector switch/E_SelectorSwitchPos.TcDUT
{attribute 'qualified_only'}
{attribute 'strict'}
{attribute 'to_string'}
TYPE E_SelectorSwitchPos :
(
	Up := 0,
	Left:=1,
	Right:=2
)BYTE;
END_TYPE

// ---- DUTs/Selector switch/ST_SelectorSwitchIO.TcDUT
TYPE ST_SelectorSwitchIO :
STRUCT
	Left	AT%I* :BIT;
	Right	AT%I* :BIT;	
END_STRUCT
END_TYPE

// ---- DUTs/Selector switch/U_SelectorSwitch.TcDUT
TYPE U_SelectorSwitch :
UNION
	IO :ST_SelectorSwitchIO;
	Pos	:E_SelectorSwitchPos;
END_UNION
END_TYPE

// ---- DUTs/ST_Point.TcDUT
TYPE ST_Point :
STRUCT
	X	:LREAL;
	Y	:LREAL;
END_STRUCT
END_TYPE

// ---- POUs/Pushbuttons/LED_Color_Enum.TcDUT
{attribute 'qualified_only'}
{attribute 'to_string'}
TYPE LED_Color_Enum :
(
	LED_RED		:= 0,
	LED_GREEN	:= 1,
	LED_BLUE	:= 2,
	LED_YELLOW	:= 3,
	LED_WHITE	:= 4
);
END_TYPE

// ---- POUs/Pushbuttons/Pushbutton_Enum.TcDUT
{attribute 'to_string'}
TYPE Pushbutton_Enum :
(
	PB_EStop	:= 0,
	PB_Start	:= 1,
	PB_Stop		:= 2,
	PB_Reset	:= 3
);
END_TYPE

// ---- POUs/MAIN.TcPOU
PROGRAM MAIN
VAR
	//SelectorSwitch			:	U_SelectorSwitch;
	//Estop					:	U_Estop;	
	Step					:	E_DemoStep;
	StartLatched			: BOOL;
	StopLatched				: BOOL;          		 	
	                		 	
	XPlanarTable  			:	FB_Component_XPlanar;
	Mover1		  			:	FB_XPlanarMover;
	Mover2		  			:	FB_XPlanarMover;
	Track1		 			:	FB_XPlanarTrackSegment;	
		            		                  		
	i						: 	UINT;
	                          	               	
	MoverStatus				:	ARRAY[1..XPlanarApplication.SystemParameters.MOVER_COUNT] OF CDT_MCTOPLC_PLANAR_MOVER_STD;
	DetectedMoversInfo		: 	XPlanarApplication.ST_TcIoMoverDetectionInfos;
							
	Mover1Target			:	ST_Point;
	Mover2Target			:	ST_Point;
	RotateTarget			:	LREAL;
	Mover1RotateTarget		:	LREAL;
	Mover2RotateTarget		:	LREAL;
	VerticalTarget			:	LREAL;
	FlipFlop				:	BOOL;
	Cycles					:	UINT;
	SubStep					:	UINT;
	                         	
	MoverCurentPos			:	ST_Point;
	
	TwinCATRestart			:	TC_Restart;
	
	rtError					:	R_TRIG;
	rtEstop					: 	R_TRIG;

	// Pushbuttons
	Init			: BOOL;
	TON_LEDFlash	: TON;
	PushButton		: ARRAY[0..3] OF FB_Pushbutton;

END_VAR                      	
VAR CONSTANT
	//Move dynamics                 	
	DEFAULT_MOVE			: 	ST_MoveDynamics := (Velocity := 500.0, 	Accel := 1000.0,	Decel := 1000.0,	Jerk := 200000.0); 
	DEFAULT_ROTATE			: 	ST_MoveDynamics := (Velocity := 5.0, 	Accel := 20.0, 		Decel := 20.0, 		Jerk := 100.0);  
	                          	
	FIGURE_EIGHT_MOVE		: 	ST_MoveDynamics := (Velocity := 750.0, 	Accel := 5000.0, 	Decel := 5000.0, 	Jerk :=200000.0);               		
	FLY_BY_MOVE				: 	ST_MoveDynamics := (Velocity := 2000.0, Accel := 20000.0, 	Decel := 20000.0, 	Jerk := 200000.0);    
	PerimeterMove			: 	ST_MoveDynamics := (Velocity := 2000.0, Accel := 20000.0, 	Decel := 20000.0, 	Jerk := 200000.0);
                              	
	ROTATE_INVERSE_MOVE		: 	ST_MoveDynamics := (Velocity := 750.0, 	Accel := 2000.0, 	Decel := 2000.0, 	Jerk := 15000.0);  
	SPIN_MOVE				: 	ST_MoveDynamics := (Velocity := 3500.0, Accel := 4000.0, 	Decel := 4000.0, 	Jerk := 20000.0);
	NUMBER_OF_SPINS			:   DINT:=30;
    
	//Move positions                         	
	START_POS_MOVER1		:	ST_Point 	:= 	(X := 60, 		Y := 60);
	START_POS_MOVER2		:	ST_Point 	:= 	(X := 180, 		Y := 180);	
	                         	
	TOP_LEFT				:	ST_POINT	:=	(X := 60.0, 	Y := 420.0);
	TOP_RIGHT				:	ST_POINT	:=	(X := 180.0, 	Y := 420.0);
	BOTTOM_LEFT				:	ST_POINT	:=	(X := 60.0, 	Y := 60.0);
	BOTTOM_RIGHT			:	ST_POINT	:=	(X := 180.0, 	Y := 60.0);
	                         	        	  	
	TOP_CENTER				:	ST_POINT	:=	(X := 120.0, 	Y := 360.0);
	BOTTOM_CENTER			:	ST_POINT	:=	(X := 120.0, 	Y := 120.0);	
END_VAR

// Cope additions to controls with Pushbuttons
PushButtonAdmin();

XplanarTable.CyclicLogic();

CASE Step OF
{region "Init"}	

	E_DemoStep.Init:
		FlipFlop		:=FALSE;
		Cycles			:=0;
		RotateTarget	:=0;
		SubStep			:=0;
		ip.Movers[1] 	:= Mover1;
		ip.Movers[2] 	:= Mover2;
		ip.Tracks[1] 	:= Track1;
		
		F_SetAllMoversMovement(DEFAULT_MOVE);
		F_SetAllMoversRotation(DEFAULT_ROTATE);

		IF XPlanarTable.InitComplete THEN
			Step			:= E_DemoStep.WaitForSwitch;
		END_IF
		
		
{endregion}
{region "WaitForSwitch"}
			
	E_DemoStep.WaitForSwitch:
		IF StartLatched THEN
			Step:= E_DemoStep.DetectMovers;
		ELSIF StopLatched THEN
			Step:= E_DemoStep.Disable;
		END_IF

		(*IF SelectorSwitch.Pos = E_SelectorSwitchPos.Left THEN
			Step:= E_DemoStep.DetectMovers;
		ELSIF SelectorSwitch.Pos = E_SelectorSwitchPos.Up THEN
			Step:= E_DemoStep.Disable;
		END_IF*)
		
{endregion}	
{region "DetectMovers"}	
	E_DemoStep.DetectMovers:
	
		IF XPlanarTable.MoverRedetect().Done THEN
			DetectedMoversInfo		:= XPlanarTable.Utility.GetMoverDetectionInfos();
			Step					:= E_DemoStep.SortMovers;
		END_IF	

{endregion}
{region "SortMovers"}	
			
	E_DemoStep.SortMovers:	
		
		IF DetectedMoversInfo.TotalDetected=2 THEN
			IF Mover1.ActualPosition.y < Mover2.ActualPosition.y THEN
				ip.Movers[1] 	:= Mover1;
				ip.Movers[2] 	:= Mover2;	
			ELSE
				ip.Movers[2] 	:= Mover1;
				ip.Movers[1] 	:= Mover2;		
			END_IF		
			Step	:= E_DemoStep.Enabling;	
		ELSIF DetectedMoversInfo.TotalDetected<>2 THEN
			Step 	:= E_DemoStep.DetectMovers;
		END_IF	

		
{endregion}	
{region "Enabling"}	

	E_DemoStep.Enabling:
		IF XplanarTable.EnableMovers().Done THEN
			Step:= E_DemoStep.SquareUpMovers;
		ELSIF XplanarTable.EnableMovers().Error THEN
			Step:= E_DemoStep.Disable;
		END_IF

	
{endregion}	
{region "SquareUpMovers"}	
	
	E_DemoStep.SquareUpMovers:	
		IF ip.Movers[1].MoveCommand.SquareUp().Done AND ip.Movers[2].MoveCommand.SquareUp().Done THEN
			Step:= E_DemoStep.MoveToSeqenceStartPos;	
		ELSIF Mover1.SquareUp().Error OR Mover2.SquareUp().Error THEN
			Step:=E_DemoStep.Disable;
		END_IF
		
{endregion}	
{region "MoveToSeqenceStartPos"}
				
	E_DemoStep.MoveToSeqenceStartPos:
		CASE SubStep OF
			0:	
				MoverCurentPos.X:=ip.Movers[1].ActualPosition.x;
				MoverCurentPos.Y:=ip.Movers[1].ActualPosition.y;
				SubStep:=1;
			1:
				IF ip.Movers[1].MoveCommand.FreeMove(MoverCurentPos.X,START_POS_MOVER1.Y).Done THEN
					SubStep:=2;
				END_IF
			2:
				IF ip.Movers[1].MoveCommand.FreeMove(START_POS_MOVER1.X,START_POS_MOVER1.Y).Done THEN
					IF ip.Movers[2].MoveCommand.FreeMove(START_POS_MOVER2.X,START_POS_MOVER2.Y).Done THEN
						SubStep	:=0;
						Step	:= E_DemoStep.JoinTrack;
					END_IF
				END_IF					
				
		END_CASE
		
{endregion}
{region "JoinTrack"}

	E_DemoStep.JoinTrack:
		IF XplanarTable.EnableTracks().Done AND 
			ip.Movers[1].MoveCommand.JoinClosestTrack(FALSE).Done AND
			ip.Movers[2].MoveCommand.JoinClosestTrack(FALSE).Done 
		THEN
			Step:= E_DemoStep.FigureEight;
			F_SetAllMoversMovement(FIGURE_EIGHT_MOVE);
		END_IF

{endregion}
{region "FigureEight"}	
	
	E_DemoStep.FigureEight:
		IF 	ip.Movers[1].MoveCommand.TrackMove(864.0+(5*Track1.TrackLength),30,Track1,Tc3_Mc3PlanarMotion.MC_DIRECTION.mcDirectionNonModulo).Done AND 
		 	ip.Movers[2].MoveCommand.TrackMove(651.0+(5*Track1.TrackLength),30,Track1,Tc3_Mc3PlanarMotion.MC_DIRECTION.mcDirectionNonModulo).Done 
		THEN
			Step:= E_DemoStep.LeaveTrack;
		END_IF
		
{endregion}
{region "LeaveTrack"}	
		
	E_DemoStep.LeaveTrack:	
		IF 	ip.Movers[1].MoveCommand.LeaveTrack(BOTTOM_LEFT.X,BOTTOM_LEFT.Y,FALSE).Done AND
			ip.Movers[2].MoveCommand.LeaveTrack(TOP_RIGHT.X,TOP_RIGHT.Y,FALSE).Done 
		THEN
			Step		:= E_DemoStep.FlyBy;
			F_SetAllMoversMovement(FLY_BY_MOVE);
			Cycles		:=0;
			FlipFlop	:=FALSE;			
		END_IF	
		
{endregion}
{region "FlyBy"}	
			
	E_DemoStep.FlyBy:		
		IF FlipFlop THEN
			Mover1Target:=TOP_LEFT;
			Mover2Target:=BOTTOM_RIGHT;
		ELSE
			Mover1Target:=BOTTOM_LEFT;
			Mover2Target:=TOP_RIGHT;				
		END_IF
		IF 	ip.Movers[1].MoveCommand.FreeMove(Mover1Target.x,Mover1Target.Y).Done AND
			ip.Movers[2].MoveCommand.FreeMove(Mover2Target.x,Mover2Target.Y).Done
		THEN
			IF FlipFlop THEN //Cycle completed
				Cycles:=Cycles+1;
				IF Cycles=4 THEN
					Step			:=E_DemoStep.MoveAroundPerimeter;
					F_SetAllMoversMovement(PerimeterMove);
					Cycles			:=0;
					SubStep			:=0;
				END_IF
			END_IF
			
			FlipFlop	:=NOT FlipFlop;
		END_IF
		
{endregion}
{region "MoveAroundPerimeter"}	

	E_DemoStep.MoveAroundPerimeter:						
		CASE SubStep OF 
			0:
				Mover1Target:=BOTTOM_LEFT;
				Mover2Target:=TOP_RIGHT;
				
			1:
				Mover1Target:=BOTTOM_RIGHT;
				Mover2Target:=TOP_LEFT;
			
			2:
				Mover1Target:=TOP_RIGHT;
				Mover2Target:=BOTTOM_LEFT;	
		
			3:
				Mover1Target:=TOP_LEFT;
				Mover2Target:=BOTTOM_RIGHT;
		END_CASE
	
		IF 	ip.Movers[1].MoveCommand.FreeMove(Mover1Target.x,Mover1Target.Y).Done AND
			ip.Movers[2].MoveCommand.FreeMove(Mover2Target.x,Mover2Target.Y).Done
		THEN
			IF SubStep=3 THEN //Cycle completed
				Cycles			:=Cycles+1;
				IF Cycles=2 THEN
					Step	:=E_DemoStep.MoveToCenterOfTiles;
				ELSE
					SubStep	:=0;
				END_IF
			ELSE
				SubStep	:=SubStep+1;
			END_IF
				
		END_IF
		
{endregion}	
{region "MoveToCenterOfTiles"}	

	E_DemoStep.MoveToCenterOfTiles:

		IF 	ip.Movers[1].MoveCommand.FreeMove(TOP_CENTER.X,TOP_CENTER.Y).Done AND
			ip.Movers[2].MoveCommand.FreeMove(BOTTOM_CENTER.X,BOTTOM_CENTER.Y).Done
		THEN
			Cycles	:=0;
			FlipFlop:=FALSE;
			Step	:=E_DemoStep.RotateInverse;
			F_SetAllMoversRotation(ROTATE_INVERSE_MOVE);
		END_IF	
		
{endregion}	
{region "RotateInverse"}	
		
	E_DemoStep.RotateInverse:
			
		IF FlipFlop THEN
			Mover1RotateTarget:=RotateTarget;
			Mover2RotateTarget:=(360.0-RotateTarget)*-1;			
		ELSE
			Mover1RotateTarget:=(360.0-RotateTarget)*-1;
			Mover2RotateTarget:=RotateTarget;
		END_IF
		
		IF 	ip.Movers[1].MoveCommand.Rotate(Mover1RotateTarget,0).Done AND
			ip.Movers[2].MoveCommand.Rotate(Mover2RotateTarget,0).Done
		THEN
			IF FlipFlop THEN
				Cycles:=Cycles+1;
				IF Cycles>=6 THEN
					Cycles		:=0;
					FlipFlop	:=FALSE;
					Step		:=E_DemoStep.Spin;
					F_SetAllMoversRotation(SPIN_MOVE);
				ELSE
					RotateTarget:=RotateTarget+15;
				END_IF
			END_IF
			FlipFlop:=NOT FlipFlop;	
		END_IF
		
{endregion}	
{region "Spin"}
		
	E_DemoStep.Spin:
	
		IF 	ip.Movers[1].MoveCommand.Rotate(0,(NUMBER_OF_SPINS*-1)).Done AND
			ip.Movers[2].MoveCommand.Rotate(0,NUMBER_OF_SPINS).Done
		THEN
			Step	:=E_DemoStep.Lift;
		END_IF		
	
{endregion}	
{region "Lift"}	

	E_DemoStep.Lift:
	
		IF FlipFlop THEN
			VerticalTarget:=2.0;
		ELSE
			VerticalTarget:=5.0;
		END_IF
		IF 	ip.Movers[1].MoveCommand.VerticalMove(VerticalTarget).Done AND
			ip.Movers[2].MoveCommand.VerticalMove(VerticalTarget).Done
		THEN
			IF FlipFlop THEN
				Cycles	:=Cycles+1;
				IF Cycles>=4 THEN
					SubStep	:=0;
					Step	:=E_DemoStep.Tilt;
				END_IF
			END_IF
			
			FlipFlop:=NOT FlipFlop;
		END_IF
	
{endregion}	
{region "Tilt"}	
	
	E_DemoStep.Tilt:
	
		CASE SubStep OF
			0:
				IF 	ip.Movers[1].MoveCommand.VerticalMove(5).Done AND
					ip.Movers[2].MoveCommand.VerticalMove(5).Done
				THEN
					SubStep:=1;
				END_IF
				
			1:
				IF 	ip.Movers[1].MoveCommand.TiltA(2).Done AND
					ip.Movers[2].MoveCommand.TiltA(-2).Done
				THEN
					SubStep:=2;
				END_IF	

			2:
			
				IF 	ip.Movers[1].MoveCommand.TiltA(-2).Done AND
					ip.Movers[2].MoveCommand.TiltA(2).Done AND
					ip.Movers[1].MoveCommand.TiltB(2).Done AND
					ip.Movers[2].MoveCommand.TiltB(-2).Done
				THEN
					SubStep:=3;
				END_IF
				
			3:	

				IF 	ip.Movers[1].MoveCommand.TiltB(-2).Done AND
					ip.Movers[2].MoveCommand.TiltB(2).Done
				THEN
					SubStep:=4;
				END_IF	
				
			4:

				IF 	ip.Movers[1].MoveCommand.TiltA(0).Done AND
					ip.Movers[2].MoveCommand.TiltA(0).Done
				THEN
					SubStep:=5;
				END_IF	

			5:
				IF 	ip.Movers[1].MoveCommand.TiltB(0).Done AND
					ip.Movers[2].MoveCommand.TiltB(0).Done
				THEN
					SubStep:=6;
				END_IF

			6:

				IF 	ip.Movers[1].MoveCommand.VerticalMove(2).Done AND
					ip.Movers[2].MoveCommand.VerticalMove(2).Done
				THEN
					Step	:=E_DemoStep.Init;
				END_IF					
				
		END_CASE
		
{endregion}			
{region "Disable"}					
    
	E_DemoStep.Disable:
	
		//Wait till the mover has completed is current move. Then disable it.
		//That way operator intervention is prevented to re-align the movers, and mover gracef
		IF NOT Mover1.Status.Busy.busyMover AND NOT Mover2.Status.Busy.busyMover THEN
			XplanarTable.DisableMovers();
		END_IF
		
		IF 	Mover1.Status.State		= MC_PLANAR_STATE.Disabled 
			AND Mover2.Status.State	= MC_PLANAR_STATE.Disabled 
			AND StartLatched
			AND NOT PushButton[PB_EStop].Pressed THEN 
 			Step:= E_DemoStep.Init;
		END_IF
		
		IF Mover1.Error THEN
			Mover1.Reset();
		END_IF
	
		IF Mover2.Error THEN
			Mover2.Reset();
		END_IF
		
		IF XPlanarTable.Error THEN
			XPlanarTable.Reset();
		END_IF
		
		IF Track1.Error THEN
			Track1.Reset();
		END_IF
		
{endregion}			
END_CASE

{region "Error detection"}

	rtError(CLK:=Mover1.Error OR Mover2.Error OR XPlanarTable.Error OR Track1.Error );
	rtEstop(CLK:=PushButton[PB_EStop].Pressed);
	IF rtError.Q OR rtEstop.Q THEN
		Step:=E_DemoStep.Disable;
	END_IF	
	
{endregion}

	
{region "Status update"}

	FOR i:=1 TO XPlanarApplication.SystemParameters.MOVER_COUNT DO
		IF ip.Movers[i]<>0 THEN		
			MoverStatus[i]:=ip.Movers[i].Status;
		END_IF
	END_FOR
	
{endregion}	


{region "System Restart"}
	//In the event of an unrecovrable error, turn the selector switch to the right
	TwinCATRestart(
		NETID:='' , 
		RESTART:= PushButton[PB_Start].Pressed AND PushButton[PB_Stop].Pressed AND PushButton[PB_Reset].Pressed);
		
{endregion}

METHOD PushButtonAdmin : BOOL
VAR_INPUT
END_VAR
// Cope additions to controls with buttons
IF NOT Init THEN
	Init							:= TRUE;
	TON_LEDFlash.PT					:= T#1S;
	PushButton[PB_EStop].LED_Color	:= LED_Color_Enum.LED_RED;
	PushButton[PB_Start].LED_Color	:= LED_Color_Enum.LED_GREEN;
	PushButton[PB_Stop].LED_Color	:= LED_Color_Enum.LED_YELLOW;
	PushButton[PB_Reset].LED_Color	:= LED_Color_Enum.LED_BLUE;
	FOR i := 0 TO 3 DO PushButton[i].rTON_Flash	REF= TON_LEDFlash; END_FOR
END_IF

// Pushbutton 
FOR i := 0 TO 3 DO
	PushButton[i]();
END_FOR

IF NOT XPlanarTable.InitComplete THEN
	FOR i := 0 TO 3 DO
		PushButton[i].Flash();
	END_FOR
	RETURN;
END_IF

TON_LEDFlash(IN := TRUE);
IF TON_LEDFlash.Q THEN
	TON_LEDFlash(IN := FALSE);
END_IF

// estop
IF PushButton[PB_EStop].Pressed THEN
	StartLatched	:= FALSE;	StopLatched	:= TRUE;
	PushButton[PB_EStop].Flash();
ELSE
	PushButton[PB_EStop].Off();
END_IF

// Start
IF PushButton[pb_start].Pressed THEN
	StartLatched	:= TRUE;	StopLatched	:= FALSE;
END_IF

IF NOT PushButton[PB_EStop].Pressed AND (Step = E_DemoStep.WaitForSwitch OR Step = E_DemoStep.Disable) THEN
	PushButton[PB_Start].Flash();
ELSIF ip.Movers[1].Status.State = MC_PLANAR_STATE.Enabled AND ip.Movers[2].Status.State = MC_PLANAR_STATE.Enabled THEN
	PushButton[PB_Start].On();
ELSE
	PushButton[PB_Start].Off();
END_IF

// Stop
IF PushButton[PB_Stop].Pressed THEN
	StartLatched	:= FALSE;	StopLatched	:= TRUE;
END_IF

IF Step = E_DemoStep.Disable AND NOT PushButton[PB_EStop].Pressed THEN
	PushButton[PB_Stop].On();
ELSIF StopLatched AND NOT PushButton[PB_EStop].Pressed THEN
	PushButton[PB_Stop].Flash();
ELSE
	PushButton[PB_Stop].Off();
END_IF

// Reset
PushButton[PB_Reset].Off();
END_METHOD

END_PROGRAM

// ---- POUs/Pushbuttons/FB_Pushbutton.TcPOU
FUNCTION_BLOCK FB_Pushbutton
VAR_INPUT
	Pressed		AT %I*	: BOOL;
	rTON_Flash	: REFERENCE TO TON;
END_VAR
VAR_OUTPUT
	LED_Red		AT %Q*	: BOOL;
	LED_Green	AT %Q*	: BOOL;
	LED_Blue	AT %Q*	: BOOL;
END_VAR
VAR
	Mode		: INT;	// 0 : OFF, 1: ON, 2: FLASH
	_LED_Color	: LED_Color_Enum;
END_VAR

CASE Mode OF
	0:	// OFF
		LED_Red		:= FALSE;
    	LED_Green	:= FALSE;
    	LED_Blue	:= FALSE;

	1,2:	// ON or Flash
		CASE _led_color OF
			LED_Color_Enum.LED_RED:
				LED_Red		:= TRUE;
				LED_Green	:= FALSE;
				LED_Blue	:= FALSE;
			LED_Color_Enum.LED_GREEN:
				LED_Red		:= FALSE;
				LED_Green	:= TRUE;
				LED_Blue	:= FALSE;
			LED_Color_Enum.LED_BLUE:
				LED_Red		:= FALSE;
				LED_Green	:= FALSE;
				LED_Blue	:= TRUE;
			LED_Color_Enum.LED_WHITE:
				LED_Red		:= TRUE;
				LED_Green	:= TRUE;
				LED_Blue	:= TRUE;
			LED_Color_Enum.LED_YELLOW:
				LED_Red		:= TRUE;
				LED_Green	:= TRUE;
				LED_Blue	:= FALSE;
		END_CASE

		// Flash
		IF Mode = 2 THEN
			LED_Red		:= LED_Red		AND rTON_Flash.ET >= rTON_Flash.PT/2;  
			LED_Green	:= LED_Green	AND rTON_Flash.ET >= rTON_Flash.PT/2;  
			LED_Blue	:= LED_Blue		AND rTON_Flash.ET >= rTON_Flash.PT/2;  
		END_IF

END_CASE

METHOD Flash : BOOL
VAR_INPUT
END_VAR
Mode	:= 2;
END_METHOD

PROPERTY LED_Color : LED_Color_Enum
GET
LED_Color	:= _LED_Color;
END_GET
SET
_LED_Color	:= LED_Color;
END_SET
END_PROPERTY

METHOD Off : BOOL
VAR_INPUT
END_VAR
Mode	:= 0;
END_METHOD

METHOD On : BOOL
VAR_INPUT
END_VAR
Mode	:= 1;
END_METHOD

END_FUNCTION_BLOCK

// ---- POUs/F_SetAllMoversMovement.TcPOU
FUNCTION F_SetAllMoversMovement : BOOL
VAR_INPUT
	Set			:ST_MoveDynamics;
END_VAR
VAR
	i			:UINT;
END_VAR

FOR i:=1 TO XPlanarApplication.SystemParameters.MOVER_COUNT DO
	IF ip.Movers[i]<>0 THEN
		ip.Movers[i].Dynamics.Movement:=Set;		
	END_IF			
END_FOR

END_FUNCTION

// ---- POUs/F_SetAllMoversRotation.TcPOU
FUNCTION F_SetAllMoversRotation : BOOL
VAR_INPUT
	Set			:ST_MoveDynamics;
END_VAR
VAR
	i			:UINT;
END_VAR

FOR i:=1 TO XPlanarApplication.SystemParameters.MOVER_COUNT DO
	IF ip.Movers[i]<>0 THEN
		ip.Movers[i].Dynamics.Rotation:=Set;		
	END_IF			
END_FOR

END_FUNCTION
